(* PLC project  *)

PROGRAM P

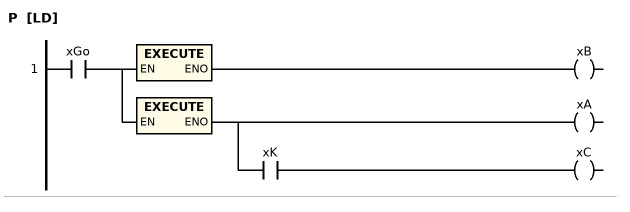
(* LD diagram, written out as Structured Text *)
IF xGo THEN
  nA := nA + 1;
END_IF;
IF xGo THEN
  nB := nB + 1;
END_IF;
xA := xGo;
xB := xGo;
xC := xGo AND xK;
END_PROGRAM
